// TIA Portal V17 export
// export: Created 2025-03-10T12:16:51.2205635Z, ExportSetting WithDefaults, DisplayName Totally Integrated Automation Portal, DisplayVersion V17 Update 8, DisplayName TIA Portal Openness, DisplayVersion V17 Update 8, DisplayName TIA Portal Version Control Interface, DisplayVersion V17, DisplayName SINAMICS Startdrive Advanced, DisplayVersion V17 SP2, DisplayName SINAMICS Startdrive G110M, G120, G120C, G120D, G120P, G115D, DisplayVersion V17 SP2, DisplayName SINAMICS Startdrive G130, G150, S120, S150, SINAMICS MV, S210, DisplayVersion V17 SP2, DisplayName STEP 7 Professional, DisplayVersion V17 Update 8, DisplayName SINUMERIK ONE STEP 7 Toolbox, DisplayVersion V17 Update 12, DisplayName SINUMERIK 840D sl STEP 7 Toolbox, DisplayVersion V17 Update 12, DisplayName STEP 7 Safety, DisplayVersion V17 Update 6, DisplayName WinCC Advanced, DisplayVersion V17 Update 8
FUNCTION "FC2392_POWER_METER" : Void   // FC2392, LAD
{ S7_Optimized_Access := 'FALSE' }
AUTHOR : ETXETAR
VERSION : 1.0
// stored: AutoNumber false, IsIECCheckEnabled false, SetENOAutomatically false, UDAEnableTagReadback false
   VAR_TEMP
      O_BYTE_0 : Struct   // OPTIONS BYTE 0
         CURRENT_UPPER_LIMIT : Bool;   // CURRENT UPPER LIMIT OPTION
         VOLTAGE_UPPER_LIMIT : Bool;   // VOLTAGE UPPER LIMIT OPTION
         VOLTAGE_LOWER_LIMIT : Bool;   // VOLTAGE LOWER LIMIT OPTION
      END_STRUCT;
      RET_VAL_1 : Int;   // RET VAL
      DATE_TIME : Date_And_Time;   // DATE AND TIME
      TOTAL_CURRENT : Real;   // TOTAL CURRENT
   END_VAR
   VAR CONSTANT
      FC_NUMBER : DInt := 2392;
   END_VAR
   VAR_TEMP   // added for the SCL form of the ladder/FBD networks
      _w1 : Bool;
      _w2 : Bool;
   END_VAR
BEGIN

REGION Network 1: OPTIONS OFF
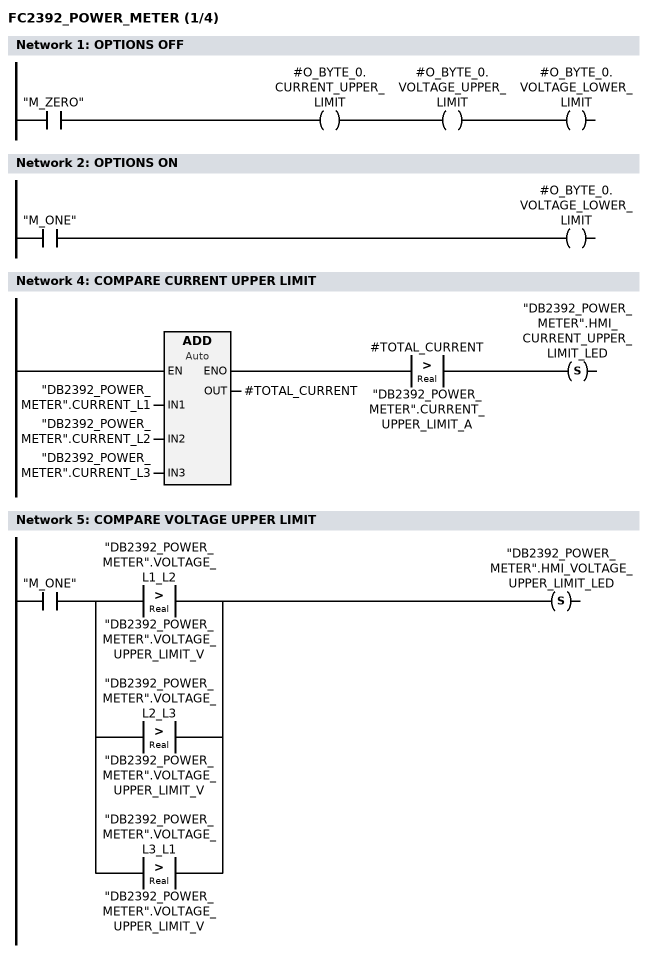
   RUNG wire#powerrail
      Contact( "M_ZERO" )
      Coil( #O_BYTE_0.CURRENT_UPPER_LIMIT )
      Coil( #O_BYTE_0.VOLTAGE_UPPER_LIMIT )
      Coil( #O_BYTE_0.VOLTAGE_LOWER_LIMIT )
   END_RUNG
   // the same network as SCL:
   #O_BYTE_0.CURRENT_UPPER_LIMIT := "M_ZERO";
   #O_BYTE_0.VOLTAGE_UPPER_LIMIT := "M_ZERO";
   #O_BYTE_0.VOLTAGE_LOWER_LIMIT := "M_ZERO";
END_REGION

REGION Network 2: OPTIONS ON
   RUNG wire#powerrail
      Contact( "M_ONE" )
      Coil( #O_BYTE_0.VOLTAGE_LOWER_LIMIT )
   END_RUNG
   // the same network as SCL:
   #O_BYTE_0.VOLTAGE_LOWER_LIMIT := "M_ONE";
END_REGION

REGION Network 3 (SCL): TRANSFER POWER METER DATA
   "DB2392_POWER_METER".VOLTAGE_L1_N := "POWER_METER_VOLTAGE_L1_N";                    //POWER METER VOLTAGE L1 N
   "DB2392_POWER_METER".VOLTAGE_L2_N := "POWER_METER_VOLTAGE_L2_N";                    //POWER METER VOLTAGE L2 N
   "DB2392_POWER_METER".VOLTAGE_L3_N := "POWER_METER_VOLTAGE_L3_N";                    //POWER METER VOLTAGE L3 N
   "DB2392_POWER_METER".VOLTAGE_L1_L2 := "POWER_METER_VOLTAGE_L1_L2";                  //POWER METER VOLTAGE L1-L2
   "DB2392_POWER_METER".VOLTAGE_L2_L3 := "POWER_METER_VOLTAGE_L2_L3";                  //POWER METER VOLTAGE L2-L3
   "DB2392_POWER_METER".VOLTAGE_L3_L1 := "POWER_METER_VOLTAGE_L3_L1";                  //POWER METER VOLTAGE L3-L1
   "DB2392_POWER_METER".CURRENT_L1 := "POWER_METER_CURRENT_L1";                        //POWER METER CURRENT L1
   "DB2392_POWER_METER".CURRENT_L2 := "POWER_METER_CURRENT_L2";                        //POWER METER CURRENT L2
   "DB2392_POWER_METER".CURRENT_L3 := "POWER_METER_CURRENT_L3";                        //POWER METER CURRENT L3
   "DB2392_POWER_METER".ACTIVE_POWER_L1 := "POWER_METER_ACTIVE_POWER_L1";              //POWER METER ACTIVE POWER L1
   "DB2392_POWER_METER".ACTIVE_POWER_L2 := "POWER_METER_ACTIVE_POWER_L2";              //POWER METER ACTIVE POWER L2
   "DB2392_POWER_METER".ACTIVE_POWER_L3 := "POWER_METER_ACTIVE_POWER_L3";              //POWER METER ACTIVE POWER L3
   "DB2392_POWER_METER".ACTIVE_ENERGY_IMPORT := "POWER_METER_ACTIVE_ENERGY_IMPORT";    //POWER METER ACTIVE ENERGY IMPORT TARRIF
   "DB2392_POWER_METER".TOTAL_ACTIVE_POWER := "POWER_METER_TOTAL_ACTIVE_POWER";        //POWER METER TOTAL ACTIVE POWER
   "DB2392_POWER_METER".TOTAL_APPARENT_FACTOR := "POWER_METER_TOTAL_APPARENT_FACTOR";  //POWER METER TOTAL APPARENT FACTOR
   "DB2392_POWER_METER".TOTAL_REACTIVE_POWER := "POWER_METER_TOTAL_REACTIVE_POWER";    //POWER METER TOTAL REACTIVE POWER
   "DB2392_POWER_METER".TOTAL_POWER_FACTOR := "POWER_METER_TOTAL_POWER_FACTOR";        //POWER METER TOTAL POWER FACTOR
   "DB2392_POWER_METER".LINE_FREQUENCY := "POWER_METER_LINE_FRECUENCY";                //POWER METER LINE FRECUENCY
END_REGION

REGION Network 4: COMPARE CURRENT UPPER LIMIT
   RUNG wire#powerrail
      Add(in1 := "DB2392_POWER_METER".CURRENT_L1, in2 := "DB2392_POWER_METER".CURRENT_L2, in3 := "DB2392_POWER_METER".CURRENT_L3, out => #TOTAL_CURRENT)
      { S7_Templates := "SrcType := Real" } GT_Contact(in1 := #TOTAL_CURRENT, in2 := "DB2392_POWER_METER".CURRENT_UPPER_LIMIT_A)
      S_Coil( "DB2392_POWER_METER".HMI_CURRENT_UPPER_LIMIT_LED )
   END_RUNG
   // the same network as SCL:
   #TOTAL_CURRENT := "DB2392_POWER_METER".CURRENT_L1 + "DB2392_POWER_METER".CURRENT_L2 + "DB2392_POWER_METER".CURRENT_L3;
   IF #TOTAL_CURRENT > "DB2392_POWER_METER".CURRENT_UPPER_LIMIT_A THEN
       "DB2392_POWER_METER".HMI_CURRENT_UPPER_LIMIT_LED := TRUE;
   END_IF;
END_REGION

REGION Network 5: COMPARE VOLTAGE UPPER LIMIT
   RUNG wire#powerrail
      Contact( "M_ONE" )
      wire#w1
      { S7_Templates := "SrcType := Real" } GT_Contact(in1 := "DB2392_POWER_METER".VOLTAGE_L1_L2, in2 := "DB2392_POWER_METER".VOLTAGE_UPPER_LIMIT_V)
      wire#w2
      S_Coil( "DB2392_POWER_METER".HMI_VOLTAGE_UPPER_LIMIT_LED )
   END_RUNG
   RUNG wire#w1
      { S7_Templates := "SrcType := Real" } GT_Contact(in1 := "DB2392_POWER_METER".VOLTAGE_L2_L3, in2 := "DB2392_POWER_METER".VOLTAGE_UPPER_LIMIT_V)
   END_RUNG wire#w2
   RUNG wire#w1
      { S7_Templates := "SrcType := Real" } GT_Contact(in1 := "DB2392_POWER_METER".VOLTAGE_L3_L1, in2 := "DB2392_POWER_METER".VOLTAGE_UPPER_LIMIT_V)
   END_RUNG wire#w2
   // the same network as SCL:
   IF "M_ONE" AND (("DB2392_POWER_METER".VOLTAGE_L1_L2 > "DB2392_POWER_METER".VOLTAGE_UPPER_LIMIT_V) OR ("DB2392_POWER_METER".VOLTAGE_L2_L3 > "DB2392_POWER_METER".VOLTAGE_UPPER_LIMIT_V) OR ("DB2392_POWER_METER".VOLTAGE_L3_L1 > "DB2392_POWER_METER".VOLTAGE_UPPER_LIMIT_V)) THEN
       "DB2392_POWER_METER".HMI_VOLTAGE_UPPER_LIMIT_LED := TRUE;
   END_IF;
END_REGION

REGION Network 6: COMPARE VOLTAGE LOWER LIMIT
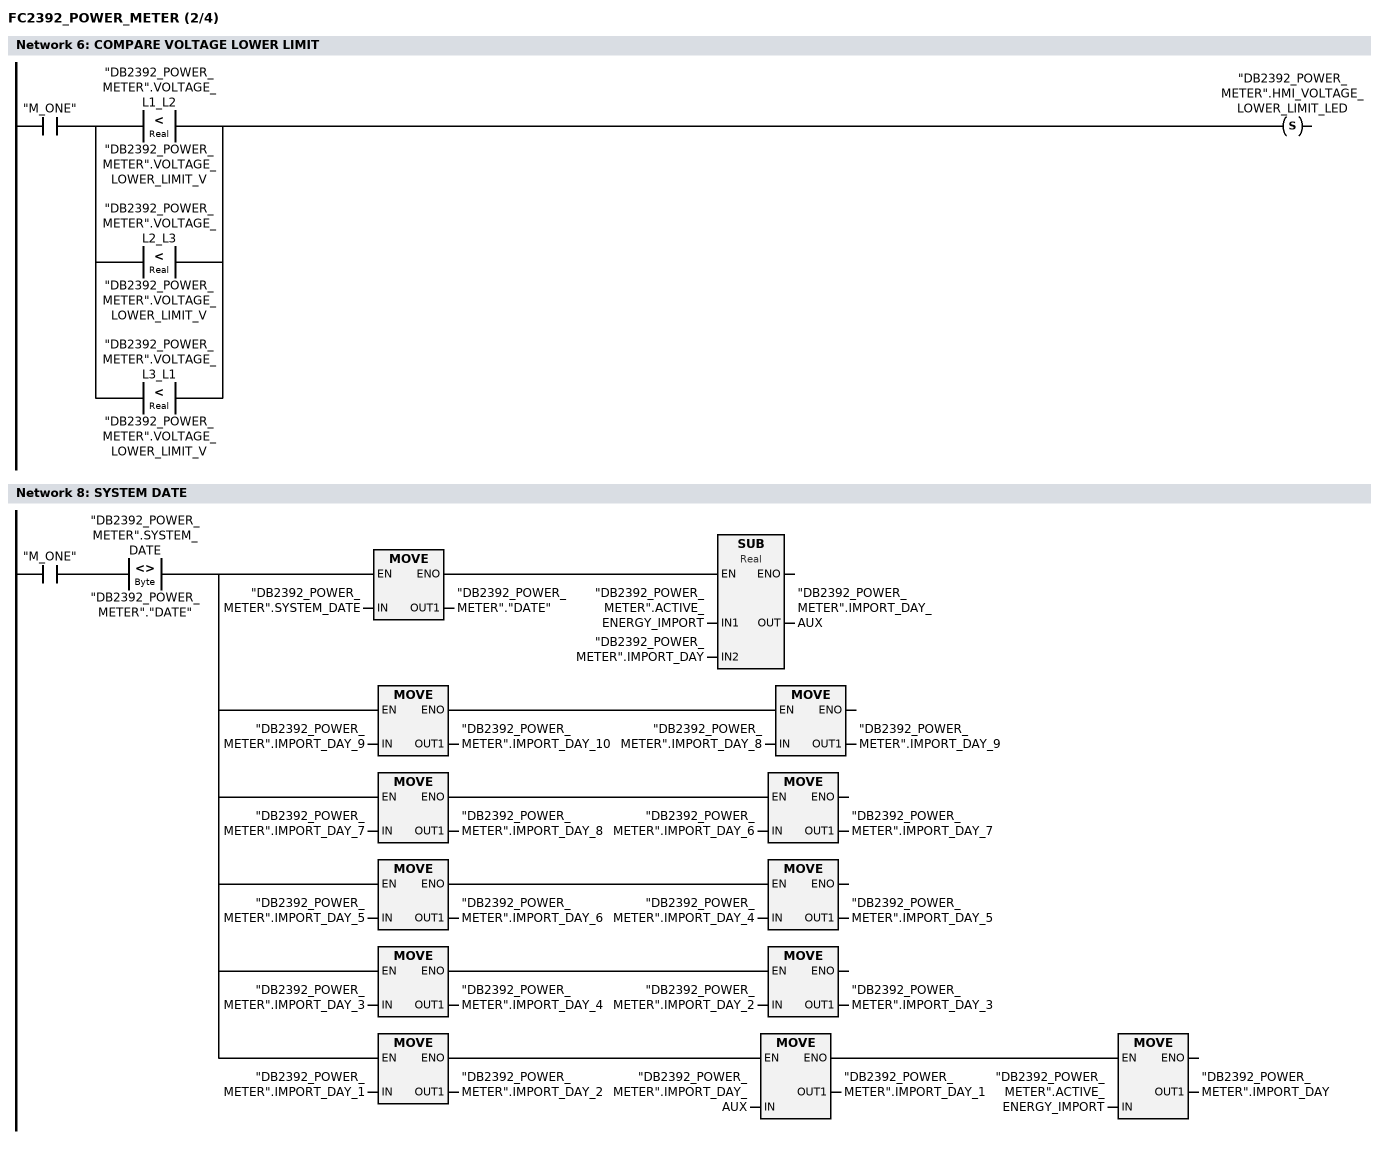
   RUNG wire#powerrail
      Contact( "M_ONE" )
      wire#w1
      { S7_Templates := "SrcType := Real" } LT_Contact(in1 := "DB2392_POWER_METER".VOLTAGE_L1_L2, in2 := "DB2392_POWER_METER".VOLTAGE_LOWER_LIMIT_V)
      wire#w2
      S_Coil( "DB2392_POWER_METER".HMI_VOLTAGE_LOWER_LIMIT_LED )
   END_RUNG
   RUNG wire#w1
      { S7_Templates := "SrcType := Real" } LT_Contact(in1 := "DB2392_POWER_METER".VOLTAGE_L2_L3, in2 := "DB2392_POWER_METER".VOLTAGE_LOWER_LIMIT_V)
   END_RUNG wire#w2
   RUNG wire#w1
      { S7_Templates := "SrcType := Real" } LT_Contact(in1 := "DB2392_POWER_METER".VOLTAGE_L3_L1, in2 := "DB2392_POWER_METER".VOLTAGE_LOWER_LIMIT_V)
   END_RUNG wire#w2
   // the same network as SCL:
   IF "M_ONE" AND (("DB2392_POWER_METER".VOLTAGE_L1_L2 < "DB2392_POWER_METER".VOLTAGE_LOWER_LIMIT_V) OR ("DB2392_POWER_METER".VOLTAGE_L2_L3 < "DB2392_POWER_METER".VOLTAGE_LOWER_LIMIT_V) OR ("DB2392_POWER_METER".VOLTAGE_L3_L1 < "DB2392_POWER_METER".VOLTAGE_LOWER_LIMIT_V)) THEN
       "DB2392_POWER_METER".HMI_VOLTAGE_LOWER_LIMIT_LED := TRUE;
   END_IF;
END_REGION

NETWORK
TITLE = READ SYSTEM TIME
      CALL  RD_SYS_T
      ( RET_VAL := #RET_VAL_1,
        OUT     := #DATE_TIME
      );
      LAR1  P##DATE_TIME;
      L     B [AR1, P#0.0];
      BTI;
      T     "DB2392_POWER_METER".SYSTEM_YEAR;
      L     B [AR1, P#1.0];
      BTI;
      T     "DB2392_POWER_METER".SYSTEM_MONTH;
      L     B [AR1, P#2.0];
      BTI;
      T     "DB2392_POWER_METER".SYSTEM_DATE;
      L     B [AR1, P#3.0];
      BTI;
      T     "DB2392_POWER_METER".SYSTEM_HOUR;
      L     B [AR1, P#4.0];
      BTI;
      T     "DB2392_POWER_METER".SYSTEM_MINUTE;
      L     B [AR1, P#5.0];
      BTI;
      T     "DB2392_POWER_METER".SYSTEM_SECOND;


REGION Network 8: SYSTEM DATE
   RUNG wire#powerrail
      Contact( "M_ONE" )
      { S7_Templates := "SrcType := Byte" } NE_Contact(in1 := "DB2392_POWER_METER".SYSTEM_DATE, in2 := "DB2392_POWER_METER"."DATE")
      wire#w1
      Move(in := "DB2392_POWER_METER".SYSTEM_DATE, out1 => "DB2392_POWER_METER"."DATE")
      { S7_Templates := "SrcType := Real" } Sub(in1 := "DB2392_POWER_METER".ACTIVE_ENERGY_IMPORT, in2 := "DB2392_POWER_METER".IMPORT_DAY, out => "DB2392_POWER_METER".IMPORT_DAY_AUX)
   END_RUNG
   RUNG wire#w1
      Move(in := "DB2392_POWER_METER".IMPORT_DAY_9, out1 => "DB2392_POWER_METER".IMPORT_DAY_10)
      Move(in := "DB2392_POWER_METER".IMPORT_DAY_8, out1 => "DB2392_POWER_METER".IMPORT_DAY_9)
   END_RUNG
   RUNG wire#w1
      Move(in := "DB2392_POWER_METER".IMPORT_DAY_7, out1 => "DB2392_POWER_METER".IMPORT_DAY_8)
      Move(in := "DB2392_POWER_METER".IMPORT_DAY_6, out1 => "DB2392_POWER_METER".IMPORT_DAY_7)
   END_RUNG
   RUNG wire#w1
      Move(in := "DB2392_POWER_METER".IMPORT_DAY_5, out1 => "DB2392_POWER_METER".IMPORT_DAY_6)
      Move(in := "DB2392_POWER_METER".IMPORT_DAY_4, out1 => "DB2392_POWER_METER".IMPORT_DAY_5)
   END_RUNG
   RUNG wire#w1
      Move(in := "DB2392_POWER_METER".IMPORT_DAY_3, out1 => "DB2392_POWER_METER".IMPORT_DAY_4)
      Move(in := "DB2392_POWER_METER".IMPORT_DAY_2, out1 => "DB2392_POWER_METER".IMPORT_DAY_3)
   END_RUNG
   RUNG wire#w1
      Move(in := "DB2392_POWER_METER".IMPORT_DAY_1, out1 => "DB2392_POWER_METER".IMPORT_DAY_2)
      Move(in := "DB2392_POWER_METER".IMPORT_DAY_AUX, out1 => "DB2392_POWER_METER".IMPORT_DAY_1)
      Move(in := "DB2392_POWER_METER".ACTIVE_ENERGY_IMPORT, out1 => "DB2392_POWER_METER".IMPORT_DAY)
   END_RUNG
   // the same network as SCL:
   #_w1 := "M_ONE" AND ("DB2392_POWER_METER".SYSTEM_DATE <> "DB2392_POWER_METER"."DATE");
   #_w2 := "M_ONE" AND ("DB2392_POWER_METER".SYSTEM_DATE <> "DB2392_POWER_METER"."DATE");
   IF #_w2 THEN
       "DB2392_POWER_METER"."DATE" := "DB2392_POWER_METER".SYSTEM_DATE;
       "DB2392_POWER_METER".IMPORT_DAY_AUX := "DB2392_POWER_METER".ACTIVE_ENERGY_IMPORT - "DB2392_POWER_METER".IMPORT_DAY;
   END_IF;
   IF #_w1 THEN
       "DB2392_POWER_METER".IMPORT_DAY_10 := "DB2392_POWER_METER".IMPORT_DAY_9;
       "DB2392_POWER_METER".IMPORT_DAY_9 := "DB2392_POWER_METER".IMPORT_DAY_8;
       "DB2392_POWER_METER".IMPORT_DAY_8 := "DB2392_POWER_METER".IMPORT_DAY_7;
       "DB2392_POWER_METER".IMPORT_DAY_7 := "DB2392_POWER_METER".IMPORT_DAY_6;
       "DB2392_POWER_METER".IMPORT_DAY_6 := "DB2392_POWER_METER".IMPORT_DAY_5;
       "DB2392_POWER_METER".IMPORT_DAY_5 := "DB2392_POWER_METER".IMPORT_DAY_4;
       "DB2392_POWER_METER".IMPORT_DAY_4 := "DB2392_POWER_METER".IMPORT_DAY_3;
       "DB2392_POWER_METER".IMPORT_DAY_3 := "DB2392_POWER_METER".IMPORT_DAY_2;
       "DB2392_POWER_METER".IMPORT_DAY_2 := "DB2392_POWER_METER".IMPORT_DAY_1;
       "DB2392_POWER_METER".IMPORT_DAY_1 := "DB2392_POWER_METER".IMPORT_DAY_AUX;
       "DB2392_POWER_METER".IMPORT_DAY := "DB2392_POWER_METER".ACTIVE_ENERGY_IMPORT;
   END_IF;
END_REGION

REGION Network 9: /////_SENTRON_PAC_/////
END_REGION

REGION Network 10: SETTINGS
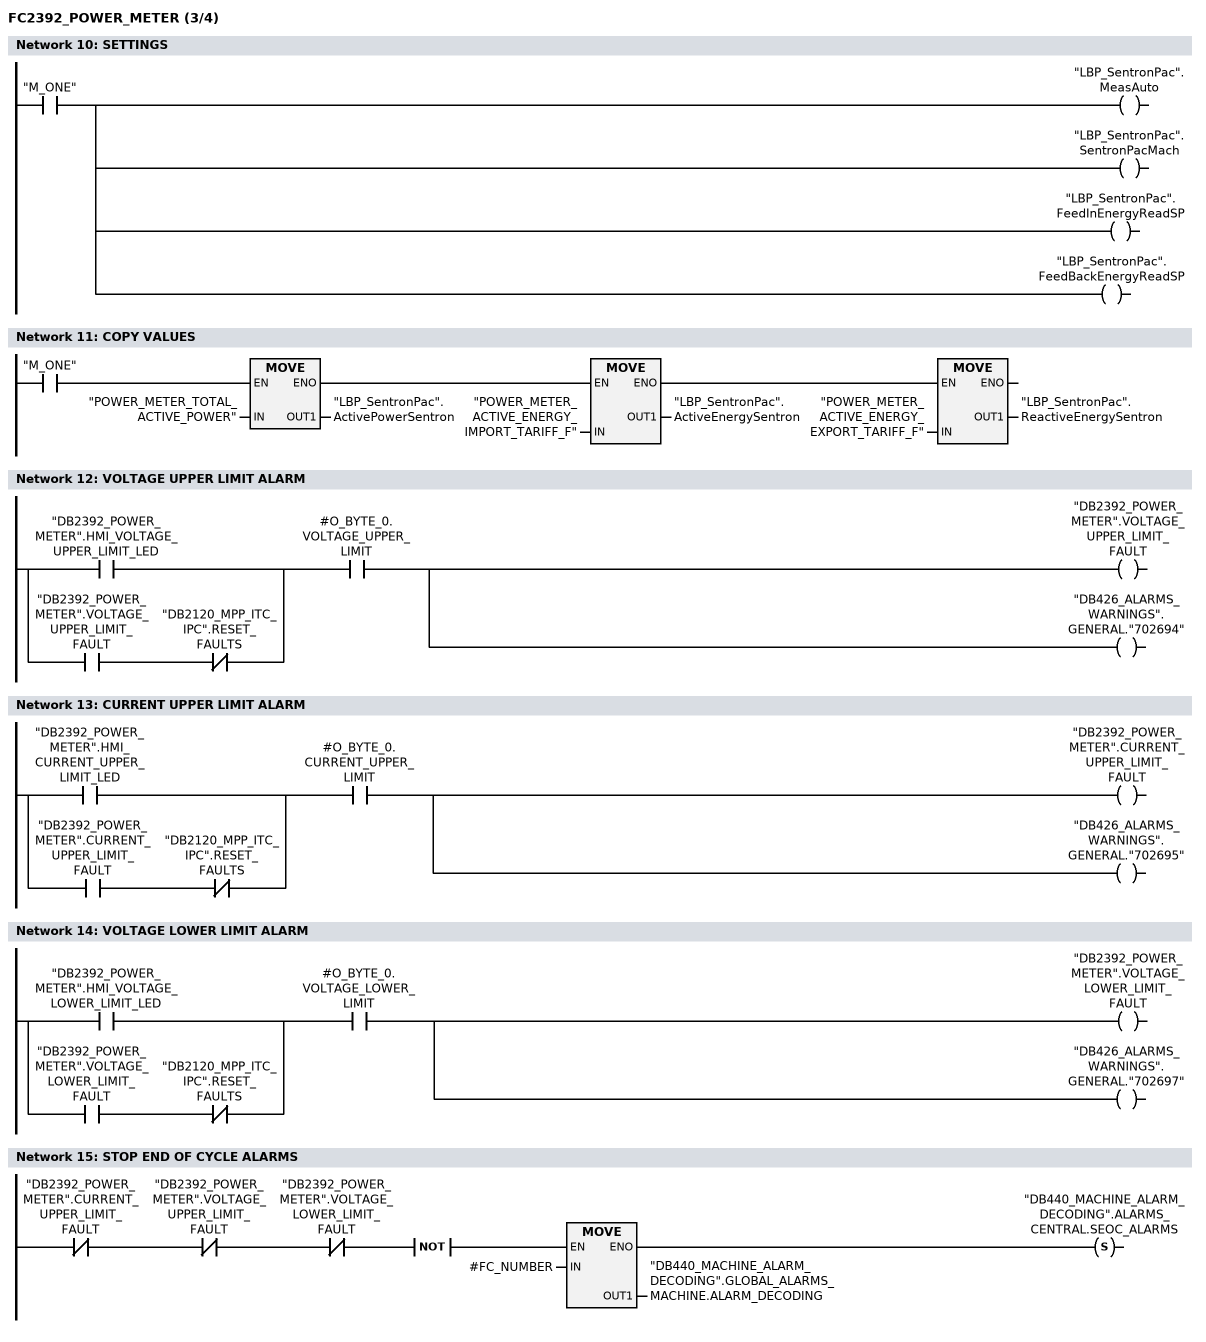
   RUNG wire#powerrail
      Contact( "M_ONE" )
      wire#w1
      Coil( "LBP_SentronPac".MeasAuto )
   END_RUNG
   RUNG wire#w1
      Coil( "LBP_SentronPac".SentronPacMach )
   END_RUNG
   RUNG wire#w1
      Coil( "LBP_SentronPac".FeedInEnergyReadSP )
   END_RUNG
   RUNG wire#w1
      Coil( "LBP_SentronPac".FeedBackEnergyReadSP )
   END_RUNG
   // the same network as SCL:
   "LBP_SentronPac".MeasAuto := "M_ONE";
   "LBP_SentronPac".SentronPacMach := "M_ONE";
   "LBP_SentronPac".FeedInEnergyReadSP := "M_ONE";
   "LBP_SentronPac".FeedBackEnergyReadSP := "M_ONE";
END_REGION

REGION Network 11: COPY VALUES
   RUNG wire#powerrail
      Contact( "M_ONE" )
      Move(in := "POWER_METER_TOTAL_ACTIVE_POWER", out1 => "LBP_SentronPac".ActivePowerSentron)
      Move(in := "POWER_METER_ACTIVE_ENERGY_IMPORT_TARIFF_F", out1 => "LBP_SentronPac".ActiveEnergySentron)
      Move(in := "POWER_METER_ACTIVE_ENERGY_EXPORT_TARIFF_F", out1 => "LBP_SentronPac".ReactiveEnergySentron)
   END_RUNG
   // the same network as SCL:
   IF "M_ONE" THEN
       "LBP_SentronPac".ActivePowerSentron := "POWER_METER_TOTAL_ACTIVE_POWER";
       "LBP_SentronPac".ActiveEnergySentron := "POWER_METER_ACTIVE_ENERGY_IMPORT_TARIFF_F";
       "LBP_SentronPac".ReactiveEnergySentron := "POWER_METER_ACTIVE_ENERGY_EXPORT_TARIFF_F";
   END_IF;
END_REGION

REGION Network 12: VOLTAGE UPPER LIMIT ALARM
   RUNG wire#powerrail
      Contact( "DB2392_POWER_METER".HMI_VOLTAGE_UPPER_LIMIT_LED )
      wire#w1
      Contact( #O_BYTE_0.VOLTAGE_UPPER_LIMIT )
      wire#w2
      Coil( "DB2392_POWER_METER".VOLTAGE_UPPER_LIMIT_FAULT )
   END_RUNG
   RUNG wire#powerrail
      Contact( "DB2392_POWER_METER".VOLTAGE_UPPER_LIMIT_FAULT )
      I_Contact( "DB2120_MPP_ITC_IPC".RESET_FAULTS )
   END_RUNG wire#w1
   RUNG wire#w2
      Coil( "DB426_ALARMS_WARNINGS".GENERAL."702694" )
   END_RUNG
   // the same network as SCL:
   "DB2392_POWER_METER".VOLTAGE_UPPER_LIMIT_FAULT := ("DB2392_POWER_METER".HMI_VOLTAGE_UPPER_LIMIT_LED OR ("DB2392_POWER_METER".VOLTAGE_UPPER_LIMIT_FAULT AND NOT "DB2120_MPP_ITC_IPC".RESET_FAULTS)) AND #O_BYTE_0.VOLTAGE_UPPER_LIMIT;
   "DB426_ALARMS_WARNINGS".GENERAL."702694" := "DB2392_POWER_METER".VOLTAGE_UPPER_LIMIT_FAULT;
END_REGION

REGION Network 13: CURRENT UPPER LIMIT ALARM
   RUNG wire#powerrail
      Contact( "DB2392_POWER_METER".HMI_CURRENT_UPPER_LIMIT_LED )
      wire#w1
      Contact( #O_BYTE_0.CURRENT_UPPER_LIMIT )
      wire#w2
      Coil( "DB2392_POWER_METER".CURRENT_UPPER_LIMIT_FAULT )
   END_RUNG
   RUNG wire#powerrail
      Contact( "DB2392_POWER_METER".CURRENT_UPPER_LIMIT_FAULT )
      I_Contact( "DB2120_MPP_ITC_IPC".RESET_FAULTS )
   END_RUNG wire#w1
   RUNG wire#w2
      Coil( "DB426_ALARMS_WARNINGS".GENERAL."702695" )
   END_RUNG
   // the same network as SCL:
   "DB2392_POWER_METER".CURRENT_UPPER_LIMIT_FAULT := ("DB2392_POWER_METER".HMI_CURRENT_UPPER_LIMIT_LED OR ("DB2392_POWER_METER".CURRENT_UPPER_LIMIT_FAULT AND NOT "DB2120_MPP_ITC_IPC".RESET_FAULTS)) AND #O_BYTE_0.CURRENT_UPPER_LIMIT;
   "DB426_ALARMS_WARNINGS".GENERAL."702695" := "DB2392_POWER_METER".CURRENT_UPPER_LIMIT_FAULT;
END_REGION

REGION Network 14: VOLTAGE LOWER LIMIT ALARM
   RUNG wire#powerrail
      Contact( "DB2392_POWER_METER".HMI_VOLTAGE_LOWER_LIMIT_LED )
      wire#w1
      Contact( #O_BYTE_0.VOLTAGE_LOWER_LIMIT )
      wire#w2
      Coil( "DB2392_POWER_METER".VOLTAGE_LOWER_LIMIT_FAULT )
   END_RUNG
   RUNG wire#powerrail
      Contact( "DB2392_POWER_METER".VOLTAGE_LOWER_LIMIT_FAULT )
      I_Contact( "DB2120_MPP_ITC_IPC".RESET_FAULTS )
   END_RUNG wire#w1
   RUNG wire#w2
      Coil( "DB426_ALARMS_WARNINGS".GENERAL."702697" )
   END_RUNG
   // the same network as SCL:
   "DB2392_POWER_METER".VOLTAGE_LOWER_LIMIT_FAULT := ("DB2392_POWER_METER".HMI_VOLTAGE_LOWER_LIMIT_LED OR ("DB2392_POWER_METER".VOLTAGE_LOWER_LIMIT_FAULT AND NOT "DB2120_MPP_ITC_IPC".RESET_FAULTS)) AND #O_BYTE_0.VOLTAGE_LOWER_LIMIT;
   "DB426_ALARMS_WARNINGS".GENERAL."702697" := "DB2392_POWER_METER".VOLTAGE_LOWER_LIMIT_FAULT;
END_REGION

REGION Network 15: STOP END OF CYCLE ALARMS
   RUNG wire#powerrail
      I_Contact( "DB2392_POWER_METER".CURRENT_UPPER_LIMIT_FAULT )
      I_Contact( "DB2392_POWER_METER".VOLTAGE_UPPER_LIMIT_FAULT )
      I_Contact( "DB2392_POWER_METER".VOLTAGE_LOWER_LIMIT_FAULT )
      Not()
      { S7_GenerateENO := "TRUE" } Move(in := #FC_NUMBER, out1 => "DB440_MACHINE_ALARM_DECODING".GLOBAL_ALARMS_MACHINE.ALARM_DECODING)
      S_Coil( "DB440_MACHINE_ALARM_DECODING".ALARMS_CENTRAL.SEOC_ALARMS )
   END_RUNG
   // the same network as SCL:
   // ENO of a box is taken as its EN; it also drops when the box reports an error
   IF NOT (NOT "DB2392_POWER_METER".CURRENT_UPPER_LIMIT_FAULT AND NOT "DB2392_POWER_METER".VOLTAGE_UPPER_LIMIT_FAULT AND NOT "DB2392_POWER_METER".VOLTAGE_LOWER_LIMIT_FAULT) THEN
       "DB440_MACHINE_ALARM_DECODING".GLOBAL_ALARMS_MACHINE.ALARM_DECODING := #FC_NUMBER;
       "DB440_MACHINE_ALARM_DECODING".ALARMS_CENTRAL.SEOC_ALARMS := TRUE;
   END_IF;
END_REGION

REGION Network 16: RESET HMI LED STATUS
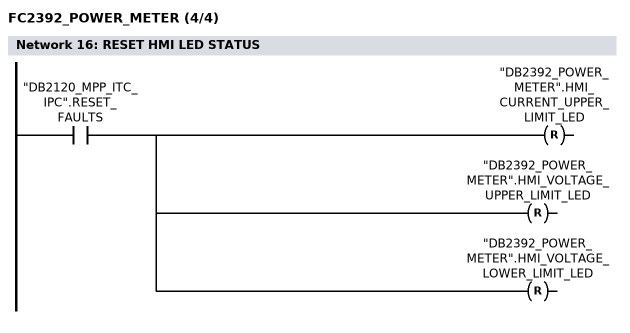
   RUNG wire#powerrail
      Contact( "DB2120_MPP_ITC_IPC".RESET_FAULTS )
      wire#w1
      R_Coil( "DB2392_POWER_METER".HMI_CURRENT_UPPER_LIMIT_LED )
   END_RUNG
   RUNG wire#w1
      R_Coil( "DB2392_POWER_METER".HMI_VOLTAGE_UPPER_LIMIT_LED )
   END_RUNG
   RUNG wire#w1
      R_Coil( "DB2392_POWER_METER".HMI_VOLTAGE_LOWER_LIMIT_LED )
   END_RUNG
   // the same network as SCL:
   IF "DB2120_MPP_ITC_IPC".RESET_FAULTS THEN
       "DB2392_POWER_METER".HMI_CURRENT_UPPER_LIMIT_LED := FALSE;
       "DB2392_POWER_METER".HMI_VOLTAGE_UPPER_LIMIT_LED := FALSE;
       "DB2392_POWER_METER".HMI_VOLTAGE_LOWER_LIMIT_LED := FALSE;
   END_IF;
END_REGION
END_FUNCTION
